// TwinCAT 3 PLC project MachineAEtat
// ProgramVersion: 3.1.4020.2
// libraries:
//   Tc2_Standard, * (Beckhoff Automation GmbH)
//   Tc2_System, * (Beckhoff Automation GmbH)
//   Tc3_Module, * (Beckhoff Automation GmbH)
// project tree:
//   / GlobalTextList.TcGTLO, PlcTask.TcTTO, Visualization Manager.TcVMO (not stored)
//   GVLs/ GVL.TcGVL
//   POUs/ MAIN.TcPOU, FB_Etape.TcPOU (not stored)
//   VISUs/ Visualization.TcVIS
// real-time tasks:
//   TASK PlcTask: cycle T#10ms, priority 20, ADS port 350

CONFIGURATION MachineAEtat
    RESOURCE PLC ON TwinCAT3
        TASK PlcTask(INTERVAL := T#10ms, PRIORITY := 20);
        PROGRAM MAIN WITH PlcTask : MAIN;
    END_RESOURCE
END_CONFIGURATION

// ---- GVLs/GVL.TcGVL
VAR_GLOBAL
	xModePasAPas :BOOL;
    xNextPas :BOOL;
END_VAR

// ---- POUs/MAIN.TcPOU
PROGRAM MAIN
VAR
	fbEtape:FB_Etape;		//step
	
END_VAR
VAR_OUTPUT
	QxLampe1 :BOOL;
	QxLampe2 :BOOL;
	QxLampe3 :BOOL;
END_VAR

(*actualisation des informations de l'objet de gestion des étapes
var 1 :gestion du blocage pour mode pas à pas
Var 2 :activation prochain pas*)
fbEtape.mActualisation(xModePasAPas,xNextPas);

CASE fbEtape.iNo OF
	//start etape
	0:	fbEtape.piVal:=100;
	
	100:fbEtape.psMess:='fonction allume lampe1';
		//assigne le temps de comptage
		fbEtape.tTimeQ:=T#1S;
		fbEtape.piVal:=110;
		
	110:fbEtape.psMess:='fonction allume lampe1';
		IF fbEtape.xTimeQ THEN
			fbEtape.piSVal:=200;
		END_IF
		
	200:fbEtape.psMess:='fonction allume lampe2';
		//assigne le nouveaux temps de comptage
		fbEtape.tTimeQ:=T#1S;
		fbEtape.piVal:=210;
		
	210:fbEtape.psMess:='fonction allume lampe2';
		IF fbEtape.xTimeQ THEN
			fbEtape.piSVal:=300;
		END_IF
		
	300:fbEtape.psMess:='fonction allume lampe3 et off lampe1';
		//assigne le nouveaux temps de comptage
		fbEtape.tTimeQ:=T#1S;
		fbEtape.piVal:=310;
		
	310:fbEtape.psMess:='fonction allume lampe3 et off lampe1';
		IF fbEtape.xTimeQ THEN
			fbEtape.piSVal:=400;
		END_IF
		
	400:fbEtape.psMess:='fonction off lampe2';
		//assigne le nouveaux temps de comptage
		fbEtape.tTimeQ:=T#1S;
		fbEtape.piVal:=410;
		
	410:fbEtape.psMess:='fonction off lampe2';
		IF fbEtape.xTimeQ THEN
			fbEtape.piSVal:=500;
		END_IF
		
	500:fbEtape.psMess:='fonction lampe 3 off';
		//assigne le nouveaux temps de comptage
		fbEtape.tTimeQ:=T#2S;
		fbEtape.piVal:=510;
		
	510:fbEtape.psMess:='fonction lampe 3 off';
		IF fbEtape.xTimeQ THEN
			fbEtape.piSVal:=100;
		END_IF
END_CASE

//--------------------------
//Actions
//--------------------------

//activation de la lampe 1
QxLampe1:=(fbEtape.iNo=110 OR fbEtape.iNo=200 OR fbEtape.iNo=210);

//activation de la lampe 2
QxLampe2:=(fbEtape.iNo=210 OR fbEtape.iNo=300 OR fbEtape.iNo=310 );

//activation de la lampe 3
QxLampe3:=(fbEtape.iNo=310 OR fbEtape.iNo=400 OR fbEtape.iNo=410) ;

END_PROGRAM

// ---- GlobalTextList.TcGTLO
TEXTLIST GlobalTextList
  1 = 'fbEtap.iNo=%i'
  0 = 'fbEtape.sMess=%s'
  2 = 'fbEtape.xTempsQ'
  3 = 'fbEtape.xTimeQ'
  4 = 'MAIN.fbEtape.xTimeQ'
END_TEXTLIST

// ---- VISUs/Visualization.TcVIS
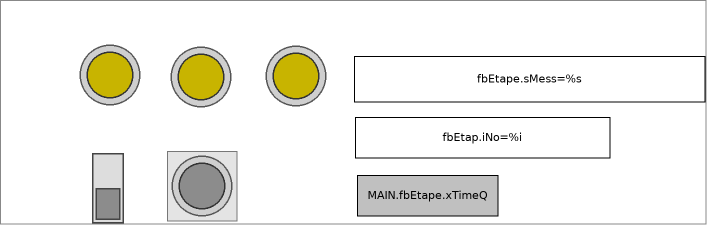
VISUALIZATION Visualization  // 707x225
    Lamp1 (75,40 70x70), variable: MAIN.QxLampe1, style: Lamp-Lamp1-Yellow
    Lamp1 (166,42 70x70), variable: MAIN.QxLampe2, style: Lamp-Lamp1-Yellow
    Lamp1 (261,41 70x70), variable: MAIN.QxLampe3, style: Lamp-Lamp1-Yellow
    DipSwitch (73,153 70x70), variable: GVL.xModePasAPas, behaviour: TOGGLE, style: Switch-DipSwitch-Gray
    PushSwitch (167,151 70x70), variable: GVL.xNextPas, behaviour: TOGGLE, style: Switch-PushSwitch-Gray
    RoundedRectangle (354,56 351x46), "fbEtape.sMess=%s", text variable: MAIN.fbEtape.sMess
    RoundedRectangle (355,117 255x41), "fbEtap.iNo=%i", text variable: MAIN.fbEtape.iNo
    RoundedRectangle (357,175 141x41), "MAIN.fbEtape.xTimeQ", colour toggle: MAIN.fbEtape.xTimeQ
END_VISUALIZATION
